FUNCTION_BLOCK RingCriticalSection (* Basic Function Block Type *)
  (* Standard: 61499-2 *)
  (* Version 0.2, 2003-12-04, JHC, Rockwell Automation, Renamed for better indexing. *)
  (* Version 0.1, 2002-11-05, JHC, Rockwell Automation, Corrected missing ST element in Algorithm REQ. *)
  (* Version 0.0, 2000-05-30, JHC, Rockwell Automation *)
  (* Compiler header: package fb.rt.cs725; *)
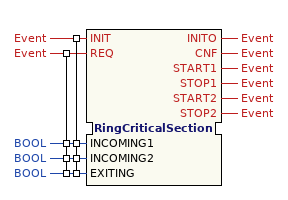
  EVENT_INPUT
    INIT WITH INCOMING1, INCOMING2, EXITING; (* Initialization Request *)
    REQ WITH INCOMING1, INCOMING2, EXITING; (* Normal Execution Request *)
  END_EVENT
  EVENT_OUTPUT
    INITO; (* Initialization Confirm *)
    CNF; (* Execution Confirmation *)
    START1;
    STOP1;
    START2;
    STOP2;
  END_EVENT
  VAR_INPUT
    INCOMING1 : BOOL; (* Input event qualifier *)
    INCOMING2 : BOOL;
    EXITING : BOOL;
  END_VAR
  VAR
    TOKEN_CLIENT : BOOL;
    TOKEN_BLOCK : BOOL;
  END_VAR
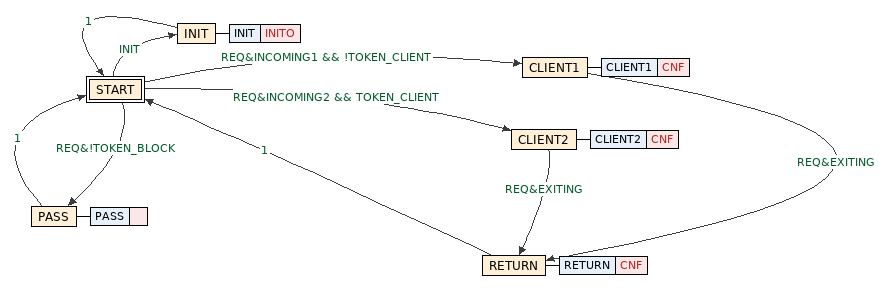
  EC_STATES
    START; (* Initial State *)
    INIT : INIT -> INITO; (* Initialization *)
    PASS : PASS; (* Normal execution *)
    CLIENT1 : CLIENT1 -> CNF;
    CLIENT2 : CLIENT2 -> CNF;
    RETURN : RETURN -> CNF;
  END_STATES
  EC_TRANSITIONS
    START TO INIT := INIT;
    INIT TO START := 1;
    START TO PASS := REQ&!TOKEN_BLOCK;
    PASS TO START := 1;
    CLIENT1 TO RETURN := REQ&EXITING;
    CLIENT2 TO RETURN := REQ&EXITING;
    RETURN TO START := 1;
    START TO CLIENT1 := REQ&INCOMING1 && !TOKEN_CLIENT;
    START TO CLIENT2 := REQ&INCOMING2 && TOKEN_CLIENT;
  END_TRANSITIONS
  ALGORITHM INIT IN ST: (* Initialization algorithm *)
TOKEN_BLOCK := FALSE;
TOKEN_CLIENT := FALSE;
  END_ALGORITHM
  ALGORITHM PASS IN ST: (* Normally executed algorithm *)
System.out.println("INCREMENTING CRITICAL: NOW " + TOKEN_CLIENT);
IF TOKEN_CLIENT THEN
TOKEN_CLIENT := FALSE;
ELSE
TOKEN_CLIENT := TRUE;
END_IF
  END_ALGORITHM
  ALGORITHM CLIENT1 IN ST:
System.out.println("CLIENT ONE HAS CRITICAL SECTION");
TOKEN_BLOCK := TRUE;
START1.serviceEvent(this);
STOP2.serviceEvent(this);
  END_ALGORITHM
  ALGORITHM CLIENT2 IN ST:
System.out.println("CLIENT TWO HAS CRITICAL SECTION");
TOKEN_BLOCK := TRUE;
STOP1.serviceEvent(this);
START2.serviceEvent(this);
  END_ALGORITHM
  ALGORITHM RETURN IN ST:
System.out.println("EXITING CRITICAL SECTION");
TOKEN_BLOCK := FALSE;
START1.serviceEvent(this);
START2.serviceEvent(this);
  END_ALGORITHM
END_FUNCTION_BLOCK
